FUNCTION_BLOCK EcMasterConfDevices IMPLEMENTS IEcTask
VAR_INPUT
END_VAR
VAR_OUTPUT
END_VAR
VAR
	iState : INT;
	masterConfDevices : Tc2_EtherCAT.FB_EcGetConfSlaves;
	_confDevices : ARRAY[0..Tc2_EtherCAT.EC_MAX_SLAVES] OF Tc2_EtherCAT.ST_EcSlaveConfigData;
	_execute: BOOL;
	_done: BOOL;
	_busy: BOOL;	
	_error: BOOL;
	_netId: AMSNETID;
END_VAR

CASE iState OF
	0:
		IF _execute THEN
			_done := FALSE;
			_busy := TRUE;
			_error := FALSE;
			masterConfDevices.bExecute := TRUE;
			IF masterConfDevices.bBusy THEN
				iState := 10;
				_execute := FALSE;
			END_IF
		END_IF
	10:
		IF NOT masterConfDevices.bBusy THEN
			IF NOT masterConfDevices.bError THEN
				_done := TRUE;
			ELSE
				_error := TRUE;
			END_IF
			_busy := FALSE;
			masterConfDevices.bExecute := FALSE;
			iState := 0;
		END_IF
END_CASE

masterConfDevices(sNetId := Tc2_System.F_CreateAmsNetId(nIds := NetId), 
					pArrEcConfSlaveInfo := ADR(_confDevices), 
					cbBufLen := SIZEOF(_confDevices));

{warning 'add method implementation '}
METHOD Abort : BOOL
masterConfDevices.bExecute := FALSE;
_busy := FALSE;
_execute := FALSE;
Abort := TRUE;
iState := 0;
END_METHOD

{warning 'add property implementation'}
PROPERTY Busy : BOOL
GET
Busy := _busy;
END_GET
END_PROPERTY

PROPERTY ConfiguredDevices : reference to array[0..Ec_Max_slaves] of St_ecslaveconfigdata
GET
ConfiguredDevices REF= _confDevices;
END_GET
END_PROPERTY

{warning 'add property implementation'}
PROPERTY Done : BOOL
GET
Done := _done;
END_GET
END_PROPERTY

{warning 'add property implementation'}
PROPERTY Error : BOOL
GET
Error := _error;
END_GET
END_PROPERTY

{warning 'add method implementation '}
METHOD Execute : BOOL
IF NOT masterConfDevices.bBusy THEN
	Execute := _execute := true;
END_IF
END_METHOD

{warning 'add property implementation'}
PROPERTY NetID : amsnetid
GET
NetID := _netId;
END_GET
SET
_netId := NetID;
END_SET
END_PROPERTY

PROPERTY NumberConfDevices : udint
GET
NumberConfDevices := masterConfDevices.nSlaves;
END_GET
END_PROPERTY

END_FUNCTION_BLOCK

(* stored: Version 1.1.0.1, ProductVersion 3.1.4024.11
   POU EcMasterConfDevices: Id {ad03dcf8-b0c6-471a-80b8-4c85c3102390}, SpecialFunc None
   Method Abort: Id {6ef9b689-653a-477d-a042-8b8bd0ce1a2c}
   Property Busy: Id {e88aedd7-5de0-44bf-89e8-8628db8cc72b}
   Get Get: Id {53562c16-68ad-498c-8bf0-5b481677b4ff}
   Property ConfiguredDevices: Id {9ef9b556-61fe-406c-94d7-18a74e07665c}
   Get Get: Id {d62b83a3-60e3-4059-9889-70bc67b43086}
   Property Done: Id {3f9a3476-d404-484f-a017-996814ae00a9}
   Get Get: Id {ace42d01-dbcf-490b-9d72-5bb0cb478ea5}
   Property Error: Id {bf1cf7da-3dc4-4146-9be8-de3d0818cf79}
   Get Get: Id {33dde674-7370-445a-acf6-293adcfb47d6}
   Method Execute: Id {5afbeb5f-7101-4271-835e-f36357f69e05}
   Property NetID: Id {650c0fc8-3dfc-479c-8788-86d3e117b7c4}
   Get Get: Id {7bdc3e21-9ece-4077-aa7e-04f2efc53788}
   Set Set: Id {a6e8fbaa-3bc5-4cd5-b73c-2760f6c26bf9}
   Property NumberConfDevices: Id {9c44f246-ced8-4dd5-a6db-f083f06e6fcf}
   Get Get: Id {47b17291-ba71-42a9-847c-86d3f9bb88a6} *)
